FUNCTION_BLOCK INTERNAL FB_SeasonStateMachine EXTENDS FB_StateMachine
VAR
    fbDefaultState:     FB_Default(THIS^, THIS^);
END_VAR

METHOD CurrentSeason : I_SeasonState
VAR_INPUT
END_VAR
__QUERYINTERFACE(THIS^.ipState, CurrentSeason);

IF CurrentSeason = 0 THEN
    CurrentSeason := THIS^.fbDefaultState;
END_IF
END_METHOD

METHOD NextSeason
VAR_INPUT
END_VAR
THIS^.CurrentSeason().NextSeason();
END_METHOD

PROPERTY StateDefault : I_SeasonState
GET
StateDefault := THIS^.fbDefaultState;
END_GET
END_PROPERTY

END_FUNCTION_BLOCK

(* stored: Version 1.1.0.1, ProductVersion 3.1.4024.12
   POU FB_SeasonStateMachine: Id {a2b4631a-918d-04a9-0d62-db5b1969a75d}, SpecialFunc None
   Method CurrentSeason: Id {45b6534a-c433-039e-0897-80c40533d81c}
   Method NextSeason: Id {55ae97dc-687b-0359-26b5-ba3cb525716c}
   Property StateDefault: Id {6853da7b-3d16-0e18-358e-858b6a5161c9}
   Get Get: Id {74dd0896-8cc0-03cc-3639-1e42fd37b648} *)
